(* Logix 5000 project; controller CLP_AB vendor 1 type 14 code 79 rev 17.4; software revision 17.01 *)

TASK DeviceNet (continuous, watchdog 500 ms) : DeviceN
TASK Initialize_speed (event, rate 10 ms, priority 10, watchdog 500 ms) : Initialize_Data
TASK MainTask (periodic, rate 50 ms, priority 10, watchdog 500 ms) : Camera_Trigger

MODULES
   Local : vendor 1 type 14 code 79 (ICP 0, rev 17.4)
      DN : vendor 1 type 12 code 14 (ICP 2, rev 7.3, Output RPI 20 ms, Input RPI 20 ms)
      Ethernet : 1756-ENBT (Ethernet 192.168.0.4, ICP 3, rev 4.1)
         Camera_Sensor : ETHERNET-MODULE (Ethernet 192.168.0.3, rev 1.1, Output RPI 25 ms)   // Banner
      LocalSERCOS : vendor 1 type 16 code 14 (ICP 1, rev 17.2, MotionAsync RPI 25 ms, MotionEvent RPI 1000 ms, MotionSync RPI 2 ms)
         Drive : vendor 1 type 115 code 164 (SERCOS 1, rev 1.1)
END_MODULES

VAR_GLOBAL   (* controller tags *)
   BitTest1 : BOOL;
   BitTest2 : BOOL;
   botao : BOOL;
   currentSpeedTopo : REAL;
   dataInitialized : BOOL;
   dir_int : DINT;
   direction : BOOL;
   drive_axis : AXIS_SERVO_DRIVE;
   dt : REAL;
   Emanuel : BOOL;
   encoder : AXIS_SERVO_DRIVE;
   IterationChange : ALIAS FOR Camera_Sensor:I.Data[6].0;
   IterationChanged : BOOL;
   IterationCount : DINT;
   lastIterationCount : DINT;
   MAH_0 : MOTION_INSTRUCTION;
   MAJ_0 : MOTION_INSTRUCTION := (FLAGS := 33554432);
   MAJ_1 : MOTION_INSTRUCTION := (FLAGS := 33554432);
   MAJ_2 : MOTION_INSTRUCTION;
   MAS_0 : MOTION_INSTRUCTION;
   MAS_1 : MOTION_INSTRUCTION := (FLAGS := 33554432);
   MAS_2 : MOTION_INSTRUCTION;
   MGroup : MOTION_GROUP;
   MSF_0 : MOTION_INSTRUCTION;
   MSO_0 : MOTION_INSTRUCTION;
   MSO_1 : MOTION_INSTRUCTION := (FLAGS := -1610612736, EN := 1, DN := 1, STATE := 1);
   OutTest1 : BOOL;
   OutTest2 : BOOL;
   position_fundo : REAL[342];
   position_topo : REAL[342];
   positionFundo : ALIAS FOR Camera_Sensor:I.Data[16];
   pyTrigger : BOOL;
   Ready : ALIAS FOR Camera_Sensor:I.Data[0].4;
   refPositionFundo : REAL;
   speed : REAL[342];
   speedRate : REAL;
   timer_1 : TIMER := (PRE := 500);
   Trigger_ACK : ALIAS FOR Camera_Sensor:I.Data[0].16;
   trigger_off : TIMER := (PRE := 10);
   trigger_on : TIMER := (PRE := 10);
END_VAR

PROGRAM Camera_Trigger   (* main routine TriggerMain *)
// Trigger
VAR
   Trigger : ALIAS FOR Camera_Sensor:O.Data[0].0;
END_VAR

ROUTINE TriggerMain   (* ladder *)
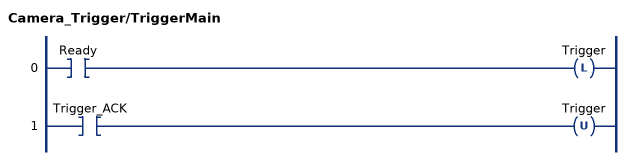
   0: XIC(Ready)OTL(Trigger);
   1: XIC(Trigger_ACK)OTU(Trigger);
END_ROUTINE
END_PROGRAM

PROGRAM Controle   (* main routine malhaAberta *)
VAR
   direcMove : DINT;
   k : DINT;
   timervel : FBD_TIMER;
END_VAR

ROUTINE ControleMain   (* structured text *)
   COP(Camera_Sensor:I.Data[6],IterationCount,32);
   if IterationCount > lastIterationCount then
   	/*Aqui vai o nosso controlador*/
   	if positionFundo > 205.0 then
   		speedRate:=.2;
   		direcMove:=1;
   	elsif positionFundo < 195.0 then
   		speedRate:=.2;
   		direcMove:=0;
   	else
   		speedRate:=0;
   		MAS(drive_axis,MAS_1,0,0,100,1,0,100,1);
   	end_if;
   	MAJ(drive_axis,MAJ_1,direcMove,speedRate,0,50.0,1,50.0,1,0,50.0,50.0,1,0,0);
   	COP(Camera_Sensor:I.Data[6],lastIterationCount,32);
   end_if;
END_ROUTINE

ROUTINE malhaAberta   (* structured text *)
   // k is the index of the speed vector
   if dataInitialized AND k < 140 then
   	currentSpeedTopo := speed[k];
   	refPositionFundo := position_fundo[k];
   	MAJ(drive_axis,MAJ_1,0,speed[k],0,50.0,1,50.0,1,0,50.0,50.0,1,0,0);
   	k:=k + 1;
   end_if;
   
   if k >= 85 then
   	MAS(drive_axis,MAS_1,0,0,100,1,0,100,1);
   	if MAS_1.DN then
   		MSF(drive_axis,MSF_0);
   	end_if;
   end_if;
END_ROUTINE

ROUTINE VeloMain   (* structured text *)
   COP(Camera_Sensor:I.Data[6],IterationCount,32);
   /*MAJ(drive_axis,MAJ_1,0,0.5,0,50.0,1,50.0,1,0,50.0,50.0,1,0,0);
   timervel.TimerEnable:=1;
   TONR(timervel);
   MAS(drive_axis,MAS_1,All,0,100,1,0,100,1);
   MSF(drive_axis,MSF_0);
   */
   	//MSO(drive_axis,MSO_1);
   	timervel.PRE:=20000;
   	if (MSO_1.EN AND timervel.ACC < 20000) then
   		if (NOT timervel.DN) then
   			timervel.TimerEnable:=1;
   			MAJ(drive_axis,MAJ_1,0,0.2,0,50.0,1,50.0,1,0,50.0,50.0,1,0,0);
   			TONR(timervel);
   		end_if;
   	end_if;
   	if (timervel.DN) then
   		MAS(drive_axis,MAS_1,All,0,100,1,0,100,1);
   	end_if;
   	if (MAS_1.EN) then
   		MSF(drive_axis,MSF_0);
   	end_if;
   
END_ROUTINE
END_PROGRAM

PROGRAM Controle1   (* main routine VeloMain *)
VAR
   direcMove : DINT;
   timervel : FBD_TIMER;
END_VAR

ROUTINE ControleMain   (* structured text *)
   COP(Camera_Sensor:I.Data[6],IterationCount,32);
   if IterationCount > lastIterationCount then
   	/*Aqui vai o nosso controlador*/
   	if positionFundo > 205.0 then
   		speedRate:=.2;
   		direcMove:=1;
   	elsif positionFundo < 195.0 then
   		speedRate:=.2;
   		direcMove:=0;
   	else
   		speedRate:=0;
   		MAS(drive_axis,MAS_1,0,0,100,1,0,100,1);
   	end_if;
   	MAJ(drive_axis,MAJ_1,direcMove,speedRate,0,50.0,1,50.0,1,0,50.0,50.0,1,0,0);
   	COP(Camera_Sensor:I.Data[6],lastIterationCount,32);
   end_if;
END_ROUTINE

ROUTINE VeloMain   (* structured text *)
   COP(Camera_Sensor:I.Data[6],IterationCount,32);
   /*MAJ(drive_axis,MAJ_1,0,0.5,0,50.0,1,50.0,1,0,50.0,50.0,1,0,0);
   timervel.TimerEnable:=1;
   TONR(timervel);
   MAS(drive_axis,MAS_1,All,0,100,1,0,100,1);
   MSF(drive_axis,MSF_0);
   */
   	//MSO(drive_axis,MSO_1);
   	timervel.PRE:=20000;
   	if (MSO_1.EN AND timervel.ACC < 20000) then
   		if (NOT timervel.DN) then
   			timervel.TimerEnable:=1;
   			MAJ(drive_axis,MAJ_1,0,0.2,0,50.0,1,50.0,1,0,50.0,50.0,1,0,0);
   			TONR(timervel);
   		end_if;
   	end_if;
   	if (timervel.DN) then
   		MAS(drive_axis,MAS_1,All,0,100,1,0,100,1);
   	end_if;
   	if (MAS_1.EN) then
   		MSF(drive_axis,MSF_0);
   	end_if;
   
END_ROUTINE
END_PROGRAM

PROGRAM DeviceN   (* main routine InitDNetST *)

ROUTINE InitDNetST   (* structured text *)
   Local:2:O.CommandRegister.Run [:=] 1;
   if (pyTrigger) AND (NOT dataInitialized) then
   	EVENT(Initialize_speed);
   end_if;
   
END_ROUTINE
END_PROGRAM

PROGRAM Initialize_Data   (* main routine Init *)

ROUTINE Init   (* structured text *)
   /* Universidade de Brasilia
   Trabalho de Graduacao em Engenharia Mecatronica
   Alunos:
   Ataias Pereira Reis 10/0093817
   Emanuel Pereira Barroso Neto 11/0115716
   This code must be executed only once. */
   
   MSO(drive_axis,MSO_1);
   
   /*Passo de tempo em segundos*/
   dt := 0.05;
   
   /*Velocidade esta em unidades/s*/
   speed[0] := 0.0;
   speed[1] := 0.0;
   speed[2] := 0.0;
   speed[3] := 0.0;
   speed[4] := 0.0;
   speed[5] := 0.0;
   speed[6] := 0.0;
   speed[7] := 0.0;
   speed[8] := 0.0;
   speed[9] := 0.0;
   speed[10] := 0.0;
   speed[11] := 0.0;
   speed[12] := 0.0;
   speed[13] := 0.0;
   speed[14] := 0.0;
   speed[15] := 0.0;
   speed[16] := 0.0;
   speed[17] := 0.0;
   speed[18] := 0.34481148756;
   speed[19] := 2.14586559751;
   speed[20] := 3.39183318828;
   speed[21] := 4.08558049026;
   speed[22] := 4.29889973402;
   speed[23] := 4.10656426872;
   speed[24] := 3.59937620076;
   speed[25] := 2.8907622351;
   speed[26] := 2.11076106434;
   speed[27] := 1.39007271596;
   speed[28] := 0.839794497606;
   speed[29] := 0.533089518345;
   speed[30] := 0.491862028501;
   speed[31] := 0.678376761817;
   speed[32] := 0.934233732939;
   speed[33] := 0.23496080216;
   speed[34] := 0.0;
   speed[35] := 0.391926043334;
   speed[36] := 1.06185403854;
   speed[37] := 1.80447758051;
   speed[38] := 2.46417142449;
   speed[39] := 2.94334148103;
   speed[40] := 3.18018087189;
   speed[41] := 3.15432700731;
   speed[42] := 2.87612098295;
   speed[43] := 2.39747816524;
   speed[44] := 1.8061682475;
   speed[45] := 1.24075219353;
   speed[46] := 0.646892038373;
   speed[47] := 0.221198064424;
   speed[48] := 0.0573516020603;
   speed[49] := 0.0;
   speed[50] := -0.0541092690492;
   speed[51] := -0.0845742147366;
   speed[52] := -0.100821711169;
   speed[53] := -0.0914084596617;
   speed[54] := -0.079105381285;
   speed[55] := 0.0;
   speed[56] := 0.0;
   speed[57] := 0.0;
   speed[58] := 0.0;
   speed[59] := 0.0;
   speed[60] := 0.0;
   speed[61] := 0.0;
   speed[62] := 0.0;
   speed[63] := 0.0;
   speed[64] := 0.0;
   speed[65] := 0.0;
   speed[66] := 0.0;
   speed[67] := 0.0;
   speed[68] := 0.0;
   speed[69] := 0.0;
   speed[70] := 0.0;
   speed[71] := 0.0;
   speed[72] := 0.0;
   speed[73] := 0.0;
   speed[74] := 0.0;
   speed[75] := 0.0;
   speed[76] := 0.0;
   speed[77] := 0.0;
   speed[78] := 0.0;
   speed[79] := 0.0;
   
   /*Posicao esta em mm*/
   position_topo[0] := 0.0;
   position_topo[1] := 0.0;
   position_topo[2] := 0.0;
   position_topo[3] := 0.0;
   position_topo[4] := 0.0;
   position_topo[5] := 0.0;
   position_topo[6] := 0.0;
   position_topo[7] := 0.0;
   position_topo[8] := 0.0;
   position_topo[9] := 0.0;
   position_topo[10] := 0.0;
   position_topo[11] := 0.0;
   position_topo[12] := 0.0;
   position_topo[13] := 0.0;
   position_topo[14] := 0.0;
   position_topo[15] := 0.0;
   position_topo[16] := 0.0;
   position_topo[17] := 0.0;
   position_topo[18] := 0.0;
   position_topo[19] := 0.00470878747236;
   position_topo[20] := 0.01475743875;
   position_topo[21] := 0.028243155676;
   position_topo[22] := 0.0433250261711;
   position_topo[23] := 0.0584203946977;
   position_topo[24] := 0.0722381619501;
   position_topo[25] := 0.0838513582337;
   position_topo[26] := 0.0927706010135;
   position_topo[27] := 0.0989769387279;
   position_topo[28] := 0.102888722485;
   position_topo[29] := 0.105257707348;
   position_topo[30] := 0.107008211828;
   position_topo[31] := 0.109038316292;
   position_topo[32] := 0.1119822507;
   position_topo[33] := 0.114128147905;
   position_topo[34] := 0.11439471649;
   position_topo[35] := 0.11500351679;
   position_topo[36] := 0.117545038466;
   position_topo[37] := 0.122660876563;
   position_topo[38] := 0.130314821323;
   position_topo[39] := 0.140022108813;
   position_topo[40] := 0.151015593143;
   position_topo[41] := 0.162387470024;
   position_topo[42] := 0.173208547671;
   position_topo[43] := 0.182658085237;
   position_topo[44] := 0.190160650649;
   position_topo[45] := 0.195649376327;
   position_topo[46] := 0.19897874828;
   position_topo[47] := 0.200457598566;
   position_topo[48] := 0.200893073888;
   position_topo[49] := 0.200980966904;
   position_topo[50] := 0.20086875201;
   position_topo[51] := 0.200616579822;
   position_topo[52] := 0.200287266523;
   position_topo[53] := 0.199949525349;
   position_topo[54] := 0.199636717374;
   position_topo[55] := 0.199414905878;
   position_topo[56] := 0.199318742002;
   position_topo[57] := 0.199298008382;
   position_topo[58] := 0.199362068337;
   position_topo[59] := 0.199451381249;
   position_topo[60] := 0.199521773358;
   position_topo[61] := 0.199560171173;
   position_topo[62] := 0.199590089344;
   position_topo[63] := 0.199602640762;
   position_topo[64] := 0.199627865053;
   position_topo[65] := 0.199632428629;
   position_topo[66] := 0.1996469843;
   position_topo[67] := 0.19966661844;
   position_topo[68] := 0.199681824736;
   position_topo[69] := 0.199703900428;
   position_topo[70] := 0.199731794629;
   position_topo[71] := 0.199761571117;
   position_topo[72] := 0.199792487952;
   position_topo[73] := 0.199828208981;
   position_topo[74] := 0.19986592834;
   position_topo[75] := 0.199898666446;
   position_topo[76] := 0.199933008111;
   position_topo[77] := 0.199967050852;
   position_topo[78] := 0.20000264005;
   position_topo[79] := 0.200039250172;
   
   position_fundo[0] := 0.0;
   position_fundo[1] := 0.0;
   position_fundo[2] := 0.0;
   position_fundo[3] := 0.0;
   position_fundo[4] := 0.0;
   position_fundo[5] := 0.0;
   position_fundo[6] := 0.0;
   position_fundo[7] := 0.0;
   position_fundo[8] := 0.0;
   position_fundo[9] := 0.0;
   position_fundo[10] := 0.0;
   position_fundo[11] := 0.0;
   position_fundo[12] := 0.0;
   position_fundo[13] := 0.0;
   position_fundo[14] := 0.0;
   position_fundo[15] := 0.0;
   position_fundo[16] := 0.0;
   position_fundo[17] := 0.0;
   position_fundo[18] := 0.0;
   position_fundo[19] := 0.0;
   position_fundo[20] := 0.0;
   position_fundo[21] := 0.0;
   position_fundo[22] := 0.0;
   position_fundo[23] := 0.0;
   position_fundo[24] := 0.0;
   position_fundo[25] := 0.0;
   position_fundo[26] := 0.0;
   position_fundo[27] := 0.00481690061308;
   position_fundo[28] := 0.0153376751732;
   position_fundo[29] := 0.0323300470963;
   position_fundo[30] := 0.0546174285514;
   position_fundo[31] := 0.0801958526907;
   position_fundo[32] := 0.106743475587;
   position_fundo[33] := 0.132028670669;
   position_fundo[34] := 0.154216668803;
   position_fundo[35] := 0.172074807259;
   position_fundo[36] := 0.185076372405;
   position_fundo[37] := 0.193402981384;
   position_fundo[38] := 0.197845574734;
   position_fundo[39] := 0.19960400628;
   position_fundo[40] := 0.19998518039;
   position_fundo[41] := 0.19999999922;
   position_fundo[42] := 0.200000000007;
   position_fundo[43] := 0.2;
   position_fundo[44] := 0.2;
   position_fundo[45] := 0.2;
   position_fundo[46] := 0.2;
   position_fundo[47] := 0.2;
   position_fundo[48] := 0.2;
   position_fundo[49] := 0.2;
   position_fundo[50] := 0.2;
   position_fundo[51] := 0.2;
   position_fundo[52] := 0.2;
   position_fundo[53] := 0.2;
   position_fundo[54] := 0.2;
   position_fundo[55] := 0.2;
   position_fundo[56] := 0.2;
   position_fundo[57] := 0.2;
   position_fundo[58] := 0.2;
   position_fundo[59] := 0.2;
   position_fundo[60] := 0.2;
   position_fundo[61] := 0.2;
   position_fundo[62] := 0.2;
   position_fundo[63] := 0.2;
   position_fundo[64] := 0.2;
   position_fundo[65] := 0.2;
   position_fundo[66] := 0.2;
   position_fundo[67] := 0.2;
   position_fundo[68] := 0.2;
   position_fundo[69] := 0.2;
   position_fundo[70] := 0.2;
   position_fundo[71] := 0.2;
   position_fundo[72] := 0.2;
   position_fundo[73] := 0.2;
   position_fundo[74] := 0.2;
   position_fundo[75] := 0.2;
   position_fundo[76] := 0.2;
   position_fundo[77] := 0.2;
   position_fundo[78] := 0.2;
   position_fundo[79] := 0.2;
   
   
   dataInitialized := 1;
   
END_ROUTINE
END_PROGRAM

PROGRAM MainProgram   (* main routine MainRoutineST *)

ROUTINE MainRoutine   (* ladder *)
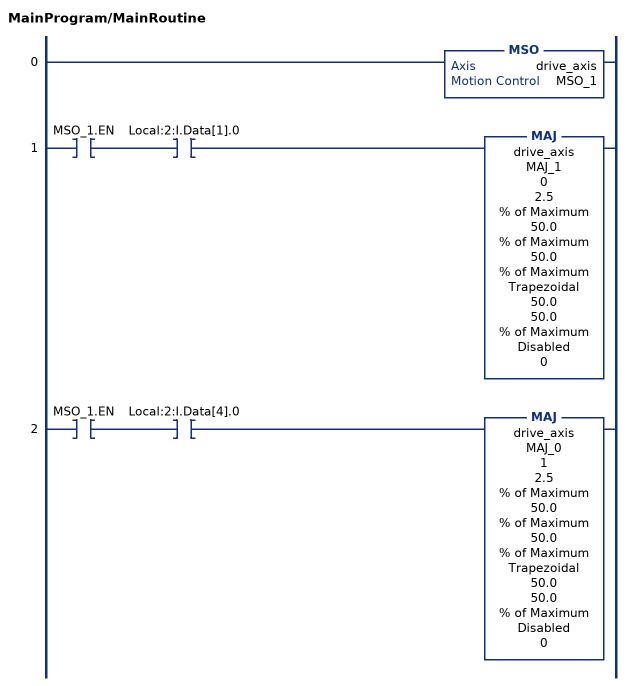
   0: MSO(drive_axis,MSO_1);
   1: XIC(MSO_1.EN)XIC(Local:2:I.Data[1].0)MAJ(drive_axis,MAJ_1,0,2.5,% of Maximum,50.0,% of Maximum,50.0,% of Maximum,Trapezoidal,50.0,50.0,% of Maximum,Disabled,0);
   2: XIC(MSO_1.EN)XIC(Local:2:I.Data[4].0)MAJ(drive_axis,MAJ_0,1,2.5,% of Maximum,50.0,% of Maximum,50.0,% of Maximum,Trapezoidal,50.0,50.0,% of Maximum,Disabled,0);
END_ROUTINE

ROUTINE MainRoutineST   (* structured text *)
   MSO(drive_axis,MSO_1);
   IF MSO_1.EN AND Local:2:I.Data[1].0 THEN
   	MAJ(drive_axis,MAJ_1,0,2.5,1,50.0,1,50.0,1,0,50.0,50.0,1,0,0);
   END_IF;
   IF MSO_1.EN AND Local:2:I.Data[4].0 THEN
   	MAJ(drive_axis,MAJ_0,1,2.5,1,50.0,1,50.0,1,0,50.0,50.0,1,0,0);
   END_IF;
END_ROUTINE
END_PROGRAM

PROGRAM Parada   (* main routine parada *)

ROUTINE parada   (* ladder *)
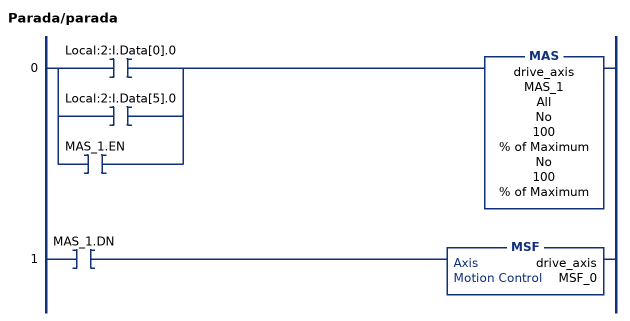
   0: [XIC(Local:2:I.Data[0].0) ,[XIC(Local:2:I.Data[5].0) ,XIC(MAS_1.EN) ] ]MAS(drive_axis,MAS_1,All,No,100,% of Maximum,No,100,% of Maximum);
   1: XIC(MAS_1.DN)MSF(drive_axis,MSF_0);
END_ROUTINE
END_PROGRAM
